(**************************************************************************************
 * 	Application		:	BoxControl Framework
 *	Revision		:	$Revision: 404529 $
 *	Revision date	:	$Date: 2018-04-23 08:21:38 +0200 (Mo., 23 Apr 2018) $
 *	Last changed by	:	$Author: b7bolm $
 *	URL				:	$URL: http://almscdc.swisslog.com/repo/SWPD/Development/BoxControlFramework/20_Release/trunk/01_Software/BCF/BCF/JumpStart/20_Product/10_App/10_Base/10_Lib/10_Conv/00_GVLs/Registry.TcGVL $
 *
 *	Purpose			:	Global registration. All types use the same
 *
 * ------------------------------------------------------------------------------------
 *	Copyright Swisslog [IP AG], Switzerland. All rights reserved.
 * 
 * ------------------------------------------------------------------------------------
 *	
 * 	Revision History: 
 *
 * 	VERSION			DATE			INITIALS			DESCRIPTION
 *	0.1				01.01.2001		swl					Example
 *
 **************************************************************************************)
VAR_GLOBAL
	FunctionRegistry	: ARRAY[E_FunctionNumber.F_BEGIN_FUNCTION..E_FunctionNumber.F_END_EXTERN_FUNCTION -1] OF ST_FunctionRegistryConv; // Function registry
	ElementRegistry 	: ARRAY[E_ElementNumber.E_BEGIN_ELEMENT..E_ElementNumber.E_END_ELEMENT -1] OF ST_ElementRegistryConv; // Element registry 
	GroupRegistry 		: ARRAY[E_GroupNumber.G_BEGIN_GROUP..E_GroupNumber.G_END_GROUP -1] OF ST_GroupRegistryConv; // Group registry 
	SubsystemRegistry	: ST_SubsystemRegistryConv; // Subsystem registry	
END_VAR

(* stored: Version 1.1.0.1, ProductVersion 3.1.4022.12
   GVL Registry: Id {150dcd13-d0fb-4f37-af19-2aa9158a87d1} *)
